# EPICS StreamDevice protocol: ioc/data/exercise5.proto
OutTerminator = LF CR
InTerminator = CR

exercise5 {

    out "DA 1"; in "1 %6i"

}
